// This function has been automatically generated from the project information.
{attribute 'signature_flag' := '1073741824'}
{attribute 'TcGenerated'}
{attribute 'no-analysis'}
FUNCTION F_GetTitle : WSTRING
VAR_INPUT
	
END_VAR

F_GetTitle := "Doc-Test";

END_FUNCTION

(* stored: Version 1.1.0.1
   POU F_GetTitle: Id {a8e65220-baa9-4b5e-8179-fea0757dc2d3}, SpecialFunc None *)
